// TIA Portal V20 export
// export: Created 2025-12-01T14:57:11.9552979Z, ExportSetting None, DisplayName Totally Integrated Automation Portal, DisplayVersion V20 Update 3, DisplayName TIA Portal Openness, DisplayVersion V20 Update 3, DisplayName TIA Portal Version Control Interface, DisplayVersion V20 Update 3, DisplayName STEP 7 Professional, DisplayVersion V20 Update 3, DisplayName STEP 7 Safety, DisplayVersion V20 Update 2, DisplayName WinCC Basic/Comfort/Advanced, DisplayVersion V20 Update 3, DisplayName WinCC Professional, DisplayVersion V20 Update 3, DisplayName WinCC Unified, DisplayVersion V20 Update 3
FUNCTION "FC771_Control_DesApiladorCajasPlastico" : Void   // FC771, STL
TITLE = Orden a generar para el Apilador de Cajas
{ S7_Optimized_Access := 'FALSE' }
AUTHOR : TRACKING
NAME : 20141014
VERSION : 4.0
// stored: AutoNumber false
   VAR_INPUT
      EstadoZonaMaquina : "EstadoZona";   // Status de la Maquina (ZONA)
      EstadoZonaMesa : "EstadoZona";   // Status de la Mesa (ZONA)
      MesaVI : UInt;   // Mesa Asociada a la Maquina
      Offset : UInt;   // Offset desde Poscion 0 hasta la Posicion Banda (+ / -)
      OrdenUT : Bool;   // Orden de Salida de la UT
      AcabadaOrden : Bool;   // Orden Acabada de la Maquina
   END_VAR
   VAR_IN_OUT
      PosInicial : UInt;   // Dato 01 de la Maquina : Posición de Recogida
      PosFinal : UInt;   // Dato 02 de la Maquina : Posición de Acabada
      TipoAmarre : UInt;   // Dato 03 de la Maquina : Tipo de Amarre
      RealizarOrden : Bool;   // Realizar la orden de la Maquina
   END_VAR
   VAR_TEMP
      NumeroUT_01 : UInt;
      NumeroUT_02 : UInt;
      NumeroUT : UInt;
      SiguienteUT : UInt;
      GrupoUT : UInt;
      AlturaF01 : UInt;
      AmarreF01 : UInt;
      AlturaF02 : UInt;
      AmarreF02 : UInt;
      CuantasUT : UInt;
   END_VAR
BEGIN

NETWORK
TITLE = Inicializaciones
/////////////////////////////////////////////////////////////////////////////
// ---  Inicializar Variables

      L     0;
      T     #AlturaF01;
      T     #AlturaF02;
      T     #AmarreF02;
      T     #CuantasUT;

      L     90;
      T     #AmarreF02;  // Por si esta vacio



NETWORK
TITLE = Reset de Variables
/////////////////////////////////////////////////////////////////////////////
// --- Si realiza un reset hay que limpiar las variables

      AN    #EstadoZonaMaquina.PerReset_CBx;
      JC    NoExiste_Reset;  // Reseteada la Maquina

      SET;
      R     #RealizarOrden;  // Resetear la orden enviada

      L     0;
      T     #PosInicial;
      T     #PosFinal;
      T     #TipoAmarre;

      JU    Final;  // Finalizado el tratamiento de la Maquina

NoExiste_Reset:NOP   0;



NETWORK
TITLE = Distribución
// - Inicialiar Variables
// - Cierre del protocolo de la orden
// - Calcular la orden
/////////////////////////////////////////////////////////////////////////////
// --- Mirar si necesita calcular orden  y cerrar protocolos

      A     #OrdenUT;
      AN    #RealizarOrden;
      AN    #AcabadaOrden;
      JC    CalcularOperacion_DelDesApilador;  // Nueva Orden a Realizar ?

      A     #AcabadaOrden;
      A     #RealizarOrden;  // Ya hay que finalizar la Orden ?
      JCN   Final;

      SET;
      R     #RealizarOrden;  // Resetear la orden enviada

      L     0;
      T     #PosInicial;
      T     #PosFinal;
      T     #TipoAmarre;

      JU    Final;  // Finalizado el tratamiento de la Maquina



NETWORK
TITLE = Calcular la Orden para la Maquina
CalcularOperacion_DelDesApilador:NOP   0;

/////////////////////////////////////////////////////////////////////////////
// --- Comprobación primera --> PosInicial, PosFinal, TipoAmarre

      L     #PosInicial;
      L     0;
      <>I;
      JC    Final;

      L     #PosFinal;
      L     0;
      <>I;
      JC    Final;

      L     #TipoAmarre;
      L     0;
      <>I;
      JC    Final;


/////////////////////////////////////////////////////////////////////////////
// --- En Marcha y sin error ==> Maquina y Mesa

      A     #EstadoZonaMaquina.Marcha_CBx;
      AN    #EstadoZonaMaquina.Error_CBx;
      A     #EstadoZonaMesa.Marcha_CBx;
      AN    #EstadoZonaMesa.Error_CBx;
      JCN   Final;


/////////////////////////////////////////////////////////////////////////////
/////////////////////////////////////////////////////////////////////////////
/////////////////////////////////////////////////////////////////////////////
// ---
// ---                  CALCULO DE LA ORDEN
// ---
/////////////////////////////////////////////////////////////////////////////
/////////////////////////////////////////////////////////////////////////////
/////////////////////////////////////////////////////////////////////////////



NETWORK
TITLE = Datos de las UT's de Mesa de Maquina
/////////////////////////////////////////////////////////////////////////////
// ---  Recoger los Datos de la Mesa de la Maquina

      L     "DB810_ColasMesas".Colas[#MesaVI].UT_PrimeraMesa;
      T     #NumeroUT;

      L     #NumeroUT;
      L     0;
      ==I;
      JC    Final;  // No hay UT's, Esta Vacia ?


/////////////////////////////////////////////////////////////////////////////
// ---  Recoger los Datos de la Primera UT de la Mesa

      L     #NumeroUT;
      T     #NumeroUT_01;

      L     "DB812_UTs_Control".UT[#NumeroUT_01].Grupo;
      T     #GrupoUT;
      L     "DB815_UTs_Datos".UT[#NumeroUT_01].CotaAltura;
      T     #AlturaF01;
      L     "DB815_UTs_Datos".UT[#NumeroUT_01].Amarre;
      T     #AmarreF01;

      L     "DB812_UTs_Control".UT[#NumeroUT_01].UT_SiguienteMesa;
      T     #SiguienteUT;

      L     #SiguienteUT;  // Solo hay Una Fila ?
      L     0;
      ==I;
      JC    Iniciar_CalculoFinal;


/////////////////////////////////////////////////////////////////////////////
// --- Datos de la siguiente UT de la Mesa en Fila Diferente

Bucle_DeBusquedaFilaSiguiente:NOP   0;
      L     #SiguienteUT;
      T     #NumeroUT_01;

      L     "DB812_UTs_Control".UT[#NumeroUT].Grupo;  // Cada Fila el Grupo es Diferente
      L     #GrupoUT;  // Hay mas de Una Fila ?
      <>I;
      JC    RecogerDatos_DeFilaSiguiente;

      L     "DB812_UTs_Control".UT[#NumeroUT].UT_SiguienteMesa;
      T     #SiguienteUT;

      L     #SiguienteUT;  // Solo hay Una Fila ?
      L     0;
      ==I;
      JC    Iniciar_CalculoFinal;
      JU    Bucle_DeBusquedaFilaSiguiente;

// --- Recoger Datos de la Segunda Fila
RecogerDatos_DeFilaSiguiente:NOP   0;
      L     #NumeroUT;
      T     #NumeroUT_02;

      L     "DB815_UTs_Datos".UT[#NumeroUT_02].CotaAltura;
      T     #AlturaF02;
      L     "DB815_UTs_Datos".UT[#NumeroUT_02].Amarre;
      T     #AmarreF02;

      L     "DB812_UTs_Control".UT[#NumeroUT_02].UT_SiguienteMesa;
      T     #NumeroUT;


/////////////////////////////////////////////////////////////////////////////
// --- Sacar tipo de Amarre, Para esta Segunda Fila
// ---         TipoAmarre = 0 - Una UT en la Fila
// ---         TipoAmarre = 1 - Dos UT en la Fila
// ---         Maximo de Dos UTs por Fila

      L     0;  // Una UT en la Fila
      T     #CuantasUT;

      L     #NumeroUT;
      L     0;
      ==I;
      JC    Iniciar_CalculoFinal;  // Es Unica en la Fila ?

      L     "DB812_UTs_Control".UT[#NumeroUT_02].Grupo;  // Cada Fila el Grupo es Diferente
      L     "DB812_UTs_Control".UT[#NumeroUT].Grupo;  // Hay una UT en la FIla
      <>I;
      JC    Iniciar_CalculoFinal;

      L     1;  // Una Dos UT's en la Fila
      T     #CuantasUT;

      JU    Iniciar_CalculoFinal;



NETWORK
TITLE = Calculo Final de Orden para la Maquina
Iniciar_CalculoFinal:NOP   0;

/////////////////////////////////////////////////////////////////////////////-
// --- Realizar el Calculo Final
// ---      Posicion Inicial
// ---      Posicion Final
// ---      Tipo de Arrarre
/////////////////////////////////////////////////////////////////////////////


/////////////////////////////////////////////////////////////////////////////
// --- Calculo de la Posicion Inicio
// ---         PosInical = AlturaF01 + AmarreF02 - 7

      L     #AlturaF01;  // AlturaF01 + AmarreF02
      L     #AmarreF02;
      +I;
      L     7;  // - 7 de Insercion de Caja
      -I;
      L     #Offset;  // + Offset de Desapilador
      +I;
      T     #PosInicial;

/////////////////////////////////////////////////////////////////////////////
// --- Calculo de la Posicion Final
// ---         PosFinal = AmarreF02 + Offset

      L     #AmarreF02;  // AmarreF02
      L     #Offset;  // + Offset de Desapilador
      +I;
      T     #PosFinal;


/////////////////////////////////////////////////////////////////////////////
// --- Calculo de la TipoAmarre
// ---         TipoAmarre = 0 - Una UT en la Fila
// ---         TipoAmarre = 1 - Dos UT en la Fila
// ---         TipoAmarre = 99 - Solo hay una Fila

      L     #CuantasUT;
      T     #TipoAmarre;

      L     #AlturaF02;
      L     0;
      <>I;
      JC    ActivarOrden;  // Es fila Unica ?

      L     99;
      T     #TipoAmarre;


/////////////////////////////////////////////////////////////////////////////
// ----------- Activacion de la Orden

ActivarOrden:SET;
      S     #RealizarOrden;
      JU    Final;



NETWORK
TITLE = Finalizar la función
/////////////////////////////////////////////////////////////////////////////
// --- Finalizado el tratamiento de la Orden
Final:NOP   0;


END_FUNCTION
